TYPE ST_Proportionair :
STRUCT
	
(* Control *)
{attribute 'pytmc' := '
        pv: Enable
        io: io
     '}
xEnable	:	BOOL;
{attribute 'pytmc' := '
        pv: Setpoint
        io: io
     '}
iSetpoint	:	INT;
{attribute 'pytmc' := '
        pv: HighLimit
        io: io
     '}
iHiLimit	:	INT;
{attribute 'pytmc' := '
        pv: LowLimit
        io: io
     '}
iLoLimit	:	INT;

(* Readback *)
xStable	: BOOL;//TTL signal from the proportionair controller that the pressure is stable
{attribute 'pytmc' := '
        pv: Pressure
        io: i
     '}
iPressure : INT;


{attribute 'TcDisplayScale' := '0-10'}
i_iPressRB AT %I* : INT;
{attribute 'TcDisplayScale' := '0-10'}
q_iPressCt AT %Q* : INT;

END_STRUCT
END_TYPE

(* stored: Version 1.1.0.1, ProductVersion 3.1.4022.18
   DUT ST_Proportionair: Id {1cb50253-0c45-4afc-8e14-284b1dbf64b6} *)
